KUKA KRL data list: Up12.dat

&ACCESS RVO1
&COMMENT VW316_7 ENTNAHME ST5085 BH2 LOW FAW RACK
&PARAM EDITMASK = Up999[1-999]
&PARAM TEMPLATE = C:\KRC\Roboter\Template\upvorgabe
&PARAM TPVW_VERSION = 8.3.17
&PARAM DISKPATH = KRC:\R1\UPs
DEFDAT Up12
; FOLD ;%{H} %MKUKATPVW
; ENDFOLD
; interface to basic routines
EXT  BAS (BAS_COMMAND  :IN,REAL  :IN )
; interface to VW-standard routines
EXT  VW (VW_COMMAND  :IN,BOOL  :IN,REAL  :IN,REAL  :IN,REAL  :IN,REAL  :IN,BOOL  :IN,E6POS  :IN )
; interface to VW_USER - Call
EXT  VW_USER (VW_USER_CMD  :IN,INT  :IN,REAL  :IN,REAL  :IN,REAL  :IN,REAL  :IN,REAL  :IN,REAL  :IN,REAL  :IN,REAL  :IN,REAL  :IN,BOOL  :IN )
EXT  VW_USR_R (VW_USER_CMD  :IN,INT  :IN,REAL  :IN,REAL  :IN,REAL  :IN,REAL  :IN,REAL  :IN,REAL  :IN,REAL  :IN,REAL  :IN,REAL  :IN,BOOL  :IN )
EXT  IBGN (IBGN_COMMAND  :IN,BOOL  :IN,REAL  :IN,REAL  :IN,BOOL  :IN,E6POS  :OUT )
; interface select routine
EXTFCT  INT  SELECT(SUBTYPE  :IN,INT  :IN,BOOL  :IN,ARI_TYP  :IN,INT  :IN,BOOL_TYP  :IN,INT  :IN,BOOL  :IN)
INT VW_NEXT_FREE=17
INT VW_NFREE_SPS=17
INT VW_MAX_SPS=117
DECL VW_MPARA_TYP P1_D={TOOL_NO 2,BASE_NO 0,VB 100,VE 0,ACC 100,TRG_TIME 5,MOVE_TYPE #PTP_MOTION}
DECL E6POS P1={X 273.551514,Y 1212.98303,Z 954.982727,A -175.620804,B 82.2778168,C -49.8938904,S 2,T 3,E1 -518.843384,E2 0.0,E3 0.0,E4 0.0,E5 0.0,E6 0.0}
DECL VW_MPARA_TYP P2_D={TOOL_NO 2,BASE_NO 0,VB 100,VE 100,ACC 100,TRG_TIME 0,MOVE_TYPE #PTP_MOTION}
DECL E6POS P2={X -689.451782,Y 1393.05701,Z 1725.33606,A 96.1449127,B 1.58781695,C 2.73405290,S 2,T 35,E1 -500.000,E2 0.0,E3 0.0,E4 0.0,E5 0.0,E6 0.0}
DECL VW_MPARA_TYP P3_D={TOOL_NO 2,BASE_NO 0,VB 100,VE 100,ACC 100,TRG_TIME 0,MOVE_TYPE #PTP_MOTION}
DECL E6POS P3={X -1311.11804,Y 1802.00903,Z 1745.52502,A 87.1430588,B 6.08077812,C -0.188109905,S 2,T 35,E1 -34.7040787,E2 0.0,E3 0.0,E4 0.0,E5 0.0,E6 0.0}
DECL VW_MPARA_TYP P4_D={TOOL_NO 2,BASE_NO 0,VB 100,VE 100,ACC 100,TRG_TIME 0,MOVE_TYPE #PTP_MOTION}
DECL E6POS P4={X -1310.30701,Y 2087.24292,Z 1150.92200,A 86.2488937,B 2.71107793,C -0.213618293,S 2,T 35,E1 -34.7040710,E2 0.0,E3 0.0,E4 0.0,E5 0.0,E6 0.0}
DECL VW_MPARA_TYP P5_D={TOOL_NO 2,BASE_NO 0,VB 100,VE 0,ACC 100,TRG_TIME 5,MOVE_TYPE #PTP_MOTION}
DECL E6POS P5={X -1308.56104,Y 2175.79492,Z 1065.74695,A 86.1406403,B 3.78117609,C -0.333399892,S 2,T 35,E1 -34.7040710,E2 0.0,E3 0.0,E4 0.0,E5 0.0,E6 0.0}
DECL VW_MPARA_TYP P6_D={TOOL_NO 2,BASE_NO 0,VB 400,VE 4711,ACC 100,TRG_TIME 5,MOVE_TYPE #GLUE_MOTION}
DECL E6POS P6={X -1314.67297,Y 2439.46509,Z 1066.40198,A 86.2557678,B 1.69427,C 0.00641007908,S 2,T 35,E1 -34.7040710,E2 0.0,E3 0.0,E4 0.0,E5 0.0,E6 0.0}
DECL VW_MPARA_TYP P7_D={TOOL_NO 2,BASE_NO 2,VB 400,VE 0,ACC 100,TRG_TIME 0,MOVE_TYPE #PATH_MOTION}
DECL E6POS P7={X 3333.12,Y 1311.37,Z 1068.54,A -3.75057602,B 1.68016100,C -0.209097296,S 2,T 35,E1 -34.7040710,E2 0.0,E3 0.0,E4 0.0,E5 0.0,E6 0.0}
DECL VW_MPARA_TYP P8_D={TOOL_NO 2,BASE_NO 31,VB 400,VE 0,ACC 100,TRG_TIME 5,MOVE_TYPE #PATH_MOTION}
DECL E6POS P8={X -58.9182281,Y -4.96595287,Z -0.879038811,A 3.90300E-06,B -2.80000E-08,C -1.31000E-07,S 2,T 35,E1 -34.7040710,E2 0.0,E3 0.0,E4 0.0,E5 0.0,E6 0.0}
DECL VW_MPARA_TYP P9_D={TOOL_NO 2,BASE_NO 31,VB 400,VE 0,ACC 100,TRG_TIME 5,MOVE_TYPE #PATH_MOTION}
DECL E6POS P9={X -94.1697388,Y -14.3363504,Z 23.2993298,A 3.84700E-06,B -5.00000E-08,C -1.39000E-07,S 2,T 35,E1 -34.7040710,E2 0.0,E3 0.0,E4 0.0,E5 0.0,E6 0.0}
DECL VW_MPARA_TYP P10_D={TOOL_NO 2,BASE_NO 0,VB 400,VE 0,ACC 100,TRG_TIME 0,MOVE_TYPE #PATH_MOTION}
DECL E6POS P10={X -1305.94971,Y 2332.87598,Z 1084.26,A 86.5534821,B 1.48964942,C 0.226125538,S 2,T 35,E1 -34.7040710,E2 0.0,E3 0.0,E4 0.0,E5 0.0,E6 0.0}
DECL VW_MPARA_TYP P11_D={TOOL_NO 2,BASE_NO 0,VB 400,VE 0,ACC 100,TRG_TIME 0,MOVE_TYPE #PATH_MOTION}
DECL E6POS P11={X -1283.60095,Y 2332.87500,Z 1200.60901,A 86.5535126,B 1.48967600,C 0.226138696,S 2,T 35,E1 -34.7040710,E2 0.0,E3 0.0,E4 0.0,E5 0.0,E6 0.0}
DECL VW_MPARA_TYP P12_D={TOOL_NO 2,BASE_NO 0,VB 400,VE 0,ACC 100,TRG_TIME 5,MOVE_TYPE #PATH_MOTION}
DECL E6POS P12={X -1283.60095,Y 2098.95288,Z 1214.83496,A 86.5535202,B 1.48967803,C 0.226144701,S 2,T 35,E1 -34.7040710,E2 0.0,E3 0.0,E4 0.0,E5 0.0,E6 0.0}
DECL VW_MPARA_TYP P13_D={TOOL_NO 2,BASE_NO 0,VB 100,VE 100,ACC 100,TRG_TIME 0,MOVE_TYPE #PTP_MOTION}
DECL E6POS P13={X -1311.11804,Y 1802.00903,Z 1745.52502,A 87.1430588,B 6.08077812,C -0.188109905,S 2,T 35,E1 -34.7040787,E2 0.0,E3 0.0,E4 0.0,E5 0.0,E6 0.0}
DECL VW_MPARA_TYP P14_D={TOOL_NO 2,BASE_NO 0,VB 100,VE 100,ACC 100,TRG_TIME 0,MOVE_TYPE #PTP_MOTION}
DECL E6POS P14={X -689.451782,Y 1393.05701,Z 1725.33606,A 96.1449127,B 1.58781695,C 2.73405290,S 2,T 35,E1 -500.000,E2 0.0,E3 0.0,E4 0.0,E5 0.0,E6 0.0}
DECL VW_MPARA_TYP P15_D={TOOL_NO 2,BASE_NO 0,VB 100,VE 100,ACC 100,TRG_TIME 0,MOVE_TYPE #PTP_MOTION}
DECL E6POS P15={X 29.5539,Y 1711.94800,Z 1336.42200,A 81.2202225,B 52.6027794,C -83.3275833,S 2,T 3,E1 -508.998688,E2 0.0,E3 0.0,E4 0.0,E5 0.0,E6 0.0}
DECL VW_MPARA_TYP P16_D={TOOL_NO 2,BASE_NO 0,VB 100,VE 0,ACC 100,TRG_TIME 5,MOVE_TYPE #PTP_MOTION}
DECL E6POS P16={X 273.551514,Y 1212.98303,Z 954.982727,A -175.620804,B 82.2778168,C -49.8938904,S 2,T 3,E1 -518.843384,E2 0.0,E3 0.0,E4 0.0,E5 0.0,E6 0.0}
ENDDAT
